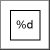
VISUALIZATION diagDPSlave  // 50x50
VAR_IN_OUT
	dataValues:typeDPSlaveIndicator;
END_VAR
    Rectangle (0,0 50x50), colour variable: dataValues.historicalState
    Rectangle (10,10 30x30), "%d", text variable: dataValues.SlaveNumber, colour variable: dataValues.currentState
END_VISUALIZATION

(* stored: Version 1.1.0.1, ProductVersion 3.1.4024.12
   Visu diagDPSlave: Id {77246471-70f4-422b-8ead-e20d301a6200} *)
